(* IEC 61131-3 sources: AXOpen/src/template.axolibrary/ctrl/src/TemplateComponent/TypesStructuresAndEnums, 5 files *)

(* ---- TemplateComponent_Component_Status.st ---- *)
NAMESPACE Template.Axolibrary
    {S7.extern=ReadWrite}
    {#ix-attr:[Container(Layout.Stack)]}
    CLASS PUBLIC TemplateComponent_Component_Status EXTENDS AXOpen.Components.Abstractions.AxoComponent_Status
        VAR PUBLIC

        END_VAR
    END_CLASS
END_NAMESPACE

(* ---- TemplateComponent_Config.st ---- *)
NAMESPACE Template.Axolibrary
    {S7.extern=ReadWrite}
    {#ix-attr:[Container(Layout.Stack)]}
    CLASS PUBLIC TemplateComponent_Config
        VAR PUBLIC
            {#ix-set:AttributeName = "<#Info time#>"}
            InfoTime : LTIME := LT#5S;
            {#ix-set:AttributeName = "<#Error time#>"}
            ErrorTime : LTIME := LT#10S;
            {#ix-set:AttributeName = "<#Task timeout#>"}
            TaskTimeout : LTIME := LT#50S;
            {#ix-set:AttributeName = "<#Hardware IDs#>"}
            HWIDs : TemplateComponent_HWIDs;
        END_VAR
    END_CLASS
END_NAMESPACE

(* ---- TemplateComponent_HWIDs.st ---- *)
NAMESPACE Template.Axolibrary
   {S7.extern=ReadWrite}
	CLASS TemplateComponent_HWIDs
      VAR PUBLIC
         {#ix-set:AttributeName = "<#Hardware ID  of the device#>"}
         HW_Device              :  UINT;
         {#ix-set:AttributeName = "<#Hardware ID of the 'in_1' submodule#>"}
         HwID_in_1            :   UINT;
         {#ix-set:AttributeName = "<#Hardware ID of the 'in_2' submodule#>"}
         HwID_in_2            :   UINT;
         {#ix-set:AttributeName = "<#Hardware ID of the 'in_3' submodule#>"}
         HwID_in_3            :   UINT;
         {#ix-set:AttributeName = "<#Hardware ID of the 'in_4' submodule#>"}
         HwID_in_4            :   UINT;
         {#ix-set:AttributeName = "<#Hardware ID of the 'in_5' submodule#>"}
         HwID_in_5            :   UINT;
         {#ix-set:AttributeName = "<#Hardware ID of the 'in_6' submodule#>"}
         HwID_in_6            :   UINT;
         {#ix-set:AttributeName = "<#Hardware ID of the 'in_7' submodule#>"}
         HwID_in_7            :   UINT;
         {#ix-set:AttributeName = "<#Hardware ID of the 'in_8' submodule#>"}
         HwID_in_8            :   UINT;
         {#ix-set:AttributeName = "<#Hardware ID of the 'in_9' submodule#>"}
         HwID_in_9            :   UINT;
         {#ix-set:AttributeName = "<#Hardware ID of the 'in_10' submodule#>"}
         HwID_in_10           :   UINT;
         {#ix-set:AttributeName = "<#Hardware ID of the 'in_11' submodule#>"}
         HwID_in_11           :   UINT;
         {#ix-set:AttributeName = "<#Hardware ID of the 'in_12' submodule#>"}
         HwID_in_12           :   UINT;
         {#ix-set:AttributeName = "<#Hardware ID of the 'in_13' submodule#>"}
         HwID_in_13           :   UINT;
         {#ix-set:AttributeName = "<#Hardware ID of the 'in_14' submodule#>"}
         HwID_in_14           :   UINT;
         {#ix-set:AttributeName = "<#Hardware ID of the 'in_15' submodule#>"}
         HwID_in_15           :   UINT;
         {#ix-set:AttributeName = "<#Hardware ID of the 'in_16' submodule#>"}
         HwID_in_16           :   UINT;
         {#ix-set:AttributeName = "<#Hardware ID of the 'in_17' submodule#>"}
         HwID_in_17           :   UINT;
         {#ix-set:AttributeName = "<#Hardware ID of the 'in_18' submodule#>"}
         HwID_in_18           :   UINT;
         {#ix-set:AttributeName = "<#Hardware ID of the 'in_19' submodule#>"}
         HwID_in_19           :   UINT;
         {#ix-set:AttributeName = "<#Hardware ID of the 'in_20' submodule#>"}
         HwID_in_20           :   UINT;
         {#ix-set:AttributeName = "<#Hardware ID of the 'out_1' submodule#>"}
         HwID_out_1           :   UINT;
         {#ix-set:AttributeName = "<#Hardware ID of the 'out_2' submodule#>"}
         HwID_out_2           :   UINT;
         {#ix-set:AttributeName = "<#Hardware ID of the 'out_3' submodule#>"}
         HwID_out_3           :   UINT;
         {#ix-set:AttributeName = "<#Hardware ID of the 'out_4' submodule#>"}
         HwID_out_4           :   UINT;
         {#ix-set:AttributeName = "<#Hardware ID of the 'out_5' submodule#>"}
         HwID_out_5           :   UINT;
         {#ix-set:AttributeName = "<#Hardware ID of the 'out_6' submodule#>"}
         HwID_out_6           :   UINT;
         {#ix-set:AttributeName = "<#Hardware ID of the 'out_7' submodule#>"}
         HwID_out_7           :   UINT;
         {#ix-set:AttributeName = "<#Hardware ID of the 'out_8' submodule#>"}
         HwID_out_8           :   UINT;
         {#ix-set:AttributeName = "<#Hardware ID of the 'out_9' submodule#>"}
         HwID_out_9           :   UINT;
         {#ix-set:AttributeName = "<#Hardware ID of the 'out_10' submodule#>"}
         HwID_out_10          :   UINT;
         {#ix-set:AttributeName = "<#Hardware ID of the 'out_11' submodule#>"}
         HwID_out_11          :   UINT;
         {#ix-set:AttributeName = "<#Hardware ID of the 'out_12' submodule#>"}
         HwID_out_12          :   UINT;
         {#ix-set:AttributeName = "<#Hardware ID of the 'out_13' submodule#>"}
         HwID_out_13          :   UINT;
         {#ix-set:AttributeName = "<#Hardware ID of the 'out_14' submodule#>"}
         HwID_out_14          :   UINT;
         {#ix-set:AttributeName = "<#Hardware ID of the 'out_15' submodule#>"}
         HwID_out_15          :   UINT;
         {#ix-set:AttributeName = "<#Hardware ID of the 'out_16' submodule#>"}
         HwID_out_16          :   UINT;
         {#ix-set:AttributeName = "<#Hardware ID of the 'out_17' submodule#>"}
         HwID_out_17          :   UINT;
         {#ix-set:AttributeName = "<#Hardware ID of the 'out_18' submodule#>"}
         HwID_out_18          :   UINT;
         {#ix-set:AttributeName = "<#Hardware ID of the 'out_19' submodule#>"}
         HwID_out_19          :   UINT;
         {#ix-set:AttributeName = "<#Hardware ID of the 'out_20' submodule#>"}
         HwID_out_20          :   UINT;
      END_VAR
   END_CLASS
END_NAMESPACE

(* ---- TemplateComponent_In.st ---- *)
NAMESPACE Template.Axolibrary
    {S7.extern=ReadWrite}
    {#ix-attr:[Container(Layout.Wrap)]}
    CLASS PUBLIC TemplateComponent_In
        VAR PUBLIC
            {#ix-set:AttributeName = "<#Status#>"}
            {#ix-attr:[ReadOnly()]}
            Status           :   TemplateComponent_Status;
        END_VAR
    END_CLASS
END_NAMESPACE

(* ---- TemplateComponent_Status.st ---- *)
NAMESPACE Template.Axolibrary
    {S7.extern=ReadWrite}
    {#ix-attr:[Container(Layout.Stack)]}
    CLASS PUBLIC TemplateComponent_Status
        VAR PUBLIC

        END_VAR
    END_CLASS
END_NAMESPACE
